REGION Network 55: STEP 1910~1940 : BDD CCV CHECK
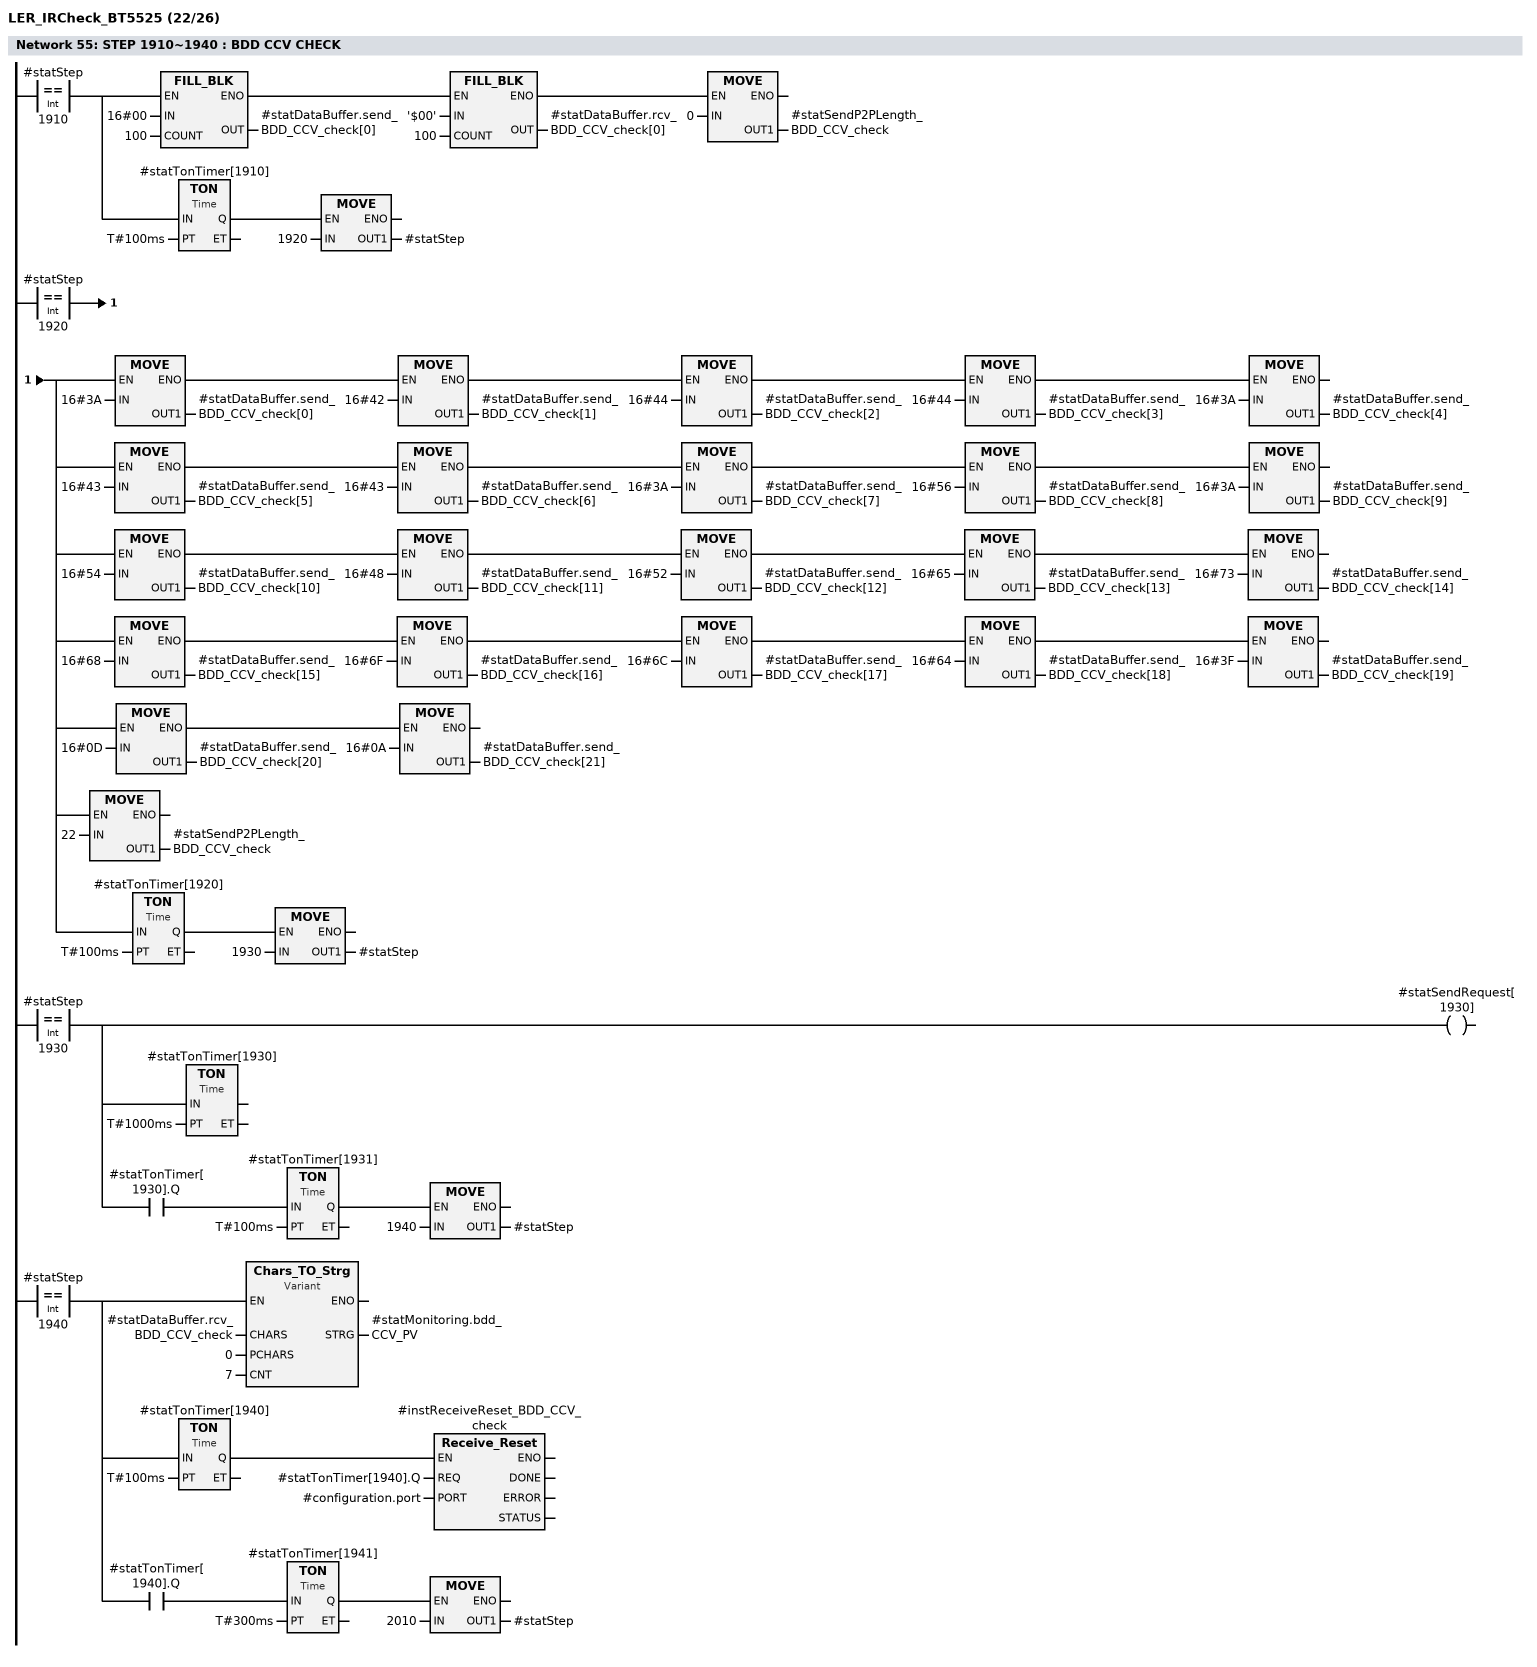
   RUNG wire#powerrail
      { S7_Templates := "SrcType := Int" } EQ_Contact(in1 := #statStep, in2 := 1910)
      wire#w1
      FillBlockI(in := 16#00, count := 100, out => #statDataBuffer.send_BDD_CCV_check[0])
      FillBlockI(in := '$00', count := 100, out => #statDataBuffer.rcv_BDD_CCV_check[0])
      Move(in := 0, out1 => #statSendP2PLength_BDD_CCV_check)
   END_RUNG
   RUNG wire#w1
      { S7_Templates := "time_type := Time" } #statTonTimer[1910].TON(pt := T#100ms, et =>)
      Move(in := 1920, out1 => #statStep)
   END_RUNG
   RUNG wire#powerrail
      { S7_Templates := "SrcType := Int" } EQ_Contact(in1 := #statStep, in2 := 1920)
      wire#w2
      Move(in := 16#3A, out1 => #statDataBuffer.send_BDD_CCV_check[0])
      Move(in := 16#42, out1 => #statDataBuffer.send_BDD_CCV_check[1])
      Move(in := 16#44, out1 => #statDataBuffer.send_BDD_CCV_check[2])
      Move(in := 16#44, out1 => #statDataBuffer.send_BDD_CCV_check[3])
      Move(in := 16#3A, out1 => #statDataBuffer.send_BDD_CCV_check[4])
   END_RUNG
   RUNG wire#w2
      Move(in := 16#43, out1 => #statDataBuffer.send_BDD_CCV_check[5])
      Move(in := 16#43, out1 => #statDataBuffer.send_BDD_CCV_check[6])
      Move(in := 16#3A, out1 => #statDataBuffer.send_BDD_CCV_check[7])
      Move(in := 16#56, out1 => #statDataBuffer.send_BDD_CCV_check[8])
      Move(in := 16#3A, out1 => #statDataBuffer.send_BDD_CCV_check[9])
   END_RUNG
   RUNG wire#w2
      Move(in := 16#54, out1 => #statDataBuffer.send_BDD_CCV_check[10])
      Move(in := 16#48, out1 => #statDataBuffer.send_BDD_CCV_check[11])
      Move(in := 16#52, out1 => #statDataBuffer.send_BDD_CCV_check[12])
      Move(in := 16#65, out1 => #statDataBuffer.send_BDD_CCV_check[13])
      Move(in := 16#73, out1 => #statDataBuffer.send_BDD_CCV_check[14])
   END_RUNG
   RUNG wire#w2
      Move(in := 16#68, out1 => #statDataBuffer.send_BDD_CCV_check[15])
      Move(in := 16#6F, out1 => #statDataBuffer.send_BDD_CCV_check[16])
      Move(in := 16#6C, out1 => #statDataBuffer.send_BDD_CCV_check[17])
      Move(in := 16#64, out1 => #statDataBuffer.send_BDD_CCV_check[18])
      Move(in := 16#3F, out1 => #statDataBuffer.send_BDD_CCV_check[19])
   END_RUNG
   RUNG wire#w2
      Move(in := 16#0D, out1 => #statDataBuffer.send_BDD_CCV_check[20])
      Move(in := 16#0A, out1 => #statDataBuffer.send_BDD_CCV_check[21])
   END_RUNG
   RUNG wire#w2
      Move(in := 22, out1 => #statSendP2PLength_BDD_CCV_check)
   END_RUNG
   RUNG wire#w2
      { S7_Templates := "time_type := Time" } #statTonTimer[1920].TON(pt := T#100ms, et =>)
      Move(in := 1930, out1 => #statStep)
   END_RUNG
   RUNG wire#powerrail
      { S7_Templates := "SrcType := Int" } EQ_Contact(in1 := #statStep, in2 := 1930)
      wire#w3
      Coil( #statSendRequest[1930] )
   END_RUNG
   RUNG wire#w3
      { S7_Templates := "time_type := Time" } #statTonTimer[1930].TON(pt := T#1000ms, et =>)
   END_RUNG
   RUNG wire#w3
      Contact( #statTonTimer[1930].Q )
      { S7_Templates := "time_type := Time" } #statTonTimer[1931].TON(pt := T#100ms, et =>)
      Move(in := 1940, out1 => #statStep)
   END_RUNG
   RUNG wire#powerrail
      { S7_Templates := "SrcType := Int" } EQ_Contact(in1 := #statStep, in2 := 1940)
      wire#w4
      { S7_Templates := "[ptr_type := Variant, str_type := String]" } Chars_TO_Strg(Chars := #statDataBuffer.rcv_BDD_CCV_check, pChars := 0, Cnt := 7, Strg => #statMonitoring.bdd_CCV_PV)
   END_RUNG
   RUNG wire#w4
      { S7_Templates := "time_type := Time" } #statTonTimer[1940].TON(pt := T#100ms, et =>)
      #instReceiveReset_BDD_CCV_check.Receive_Reset(REQ := #statTonTimer[1940].Q, PORT := #configuration.port, DONE =>, ERROR =>, STATUS =>)
   END_RUNG
   RUNG wire#w4
      Contact( #statTonTimer[1940].Q )
      { S7_Templates := "time_type := Time" } #statTonTimer[1941].TON(pt := T#300ms, et =>)
      Move(in := 2010, out1 => #statStep)
   END_RUNG
   // the same network as SCL:
   #_w1 := #statStep = 1910;
   IF #_w1 THEN
       FILL_BLK(IN := 16#00, COUNT := 100, OUT => #statDataBuffer.send_BDD_CCV_check[0]);
       FILL_BLK(IN := '$00', COUNT := 100, OUT => #statDataBuffer.rcv_BDD_CCV_check[0]);
       #statSendP2PLength_BDD_CCV_check := 0;
   END_IF;
   #statTonTimer[1910].TON(IN := #_w1, PT := T#100ms);
   IF #statTonTimer[1910].Q THEN #statStep := 1920; END_IF;
   #_w2 := #statStep = 1920;
   IF #_w2 THEN
       #statDataBuffer.send_BDD_CCV_check[0] := 16#3A;
       #statDataBuffer.send_BDD_CCV_check[1] := 16#42;
       #statDataBuffer.send_BDD_CCV_check[2] := 16#44;
       #statDataBuffer.send_BDD_CCV_check[3] := 16#44;
       #statDataBuffer.send_BDD_CCV_check[4] := 16#3A;
       #statDataBuffer.send_BDD_CCV_check[5] := 16#43;
       #statDataBuffer.send_BDD_CCV_check[6] := 16#43;
       #statDataBuffer.send_BDD_CCV_check[7] := 16#3A;
       #statDataBuffer.send_BDD_CCV_check[8] := 16#56;
       #statDataBuffer.send_BDD_CCV_check[9] := 16#3A;
       #statDataBuffer.send_BDD_CCV_check[10] := 16#54;
       #statDataBuffer.send_BDD_CCV_check[11] := 16#48;
       #statDataBuffer.send_BDD_CCV_check[12] := 16#52;
       #statDataBuffer.send_BDD_CCV_check[13] := 16#65;
       #statDataBuffer.send_BDD_CCV_check[14] := 16#73;
       #statDataBuffer.send_BDD_CCV_check[15] := 16#68;
       #statDataBuffer.send_BDD_CCV_check[16] := 16#6F;
       #statDataBuffer.send_BDD_CCV_check[17] := 16#6C;
       #statDataBuffer.send_BDD_CCV_check[18] := 16#64;
       #statDataBuffer.send_BDD_CCV_check[19] := 16#3F;
       #statDataBuffer.send_BDD_CCV_check[20] := 16#0D;
       #statDataBuffer.send_BDD_CCV_check[21] := 16#0A;
       #statSendP2PLength_BDD_CCV_check := 22;
   END_IF;
   #statTonTimer[1920].TON(IN := #_w2, PT := T#100ms);
   IF #statTonTimer[1920].Q THEN #statStep := 1930; END_IF;
   #statSendRequest[1930] := #statStep = 1930;
   #statTonTimer[1930].TON(IN := #statStep = 1930, PT := T#1000ms);
   #statTonTimer[1931].TON(IN := (#statStep = 1930) AND #statTonTimer[1930].Q, PT := T#100ms);
   IF #statTonTimer[1931].Q THEN #statStep := 1940; END_IF;
   #_w3 := #statStep = 1940;
   IF #_w3 THEN
       Chars_TO_Strg(Chars := #statDataBuffer.rcv_BDD_CCV_check,
                     pChars := 0,
                     Cnt := 7,
                     Strg => #statMonitoring.bdd_CCV_PV);
   END_IF;
   #statTonTimer[1940].TON(IN := #_w3, PT := T#100ms);
   IF #statTonTimer[1940].Q THEN
       #instReceiveReset_BDD_CCV_check(REQ := #statTonTimer[1940].Q, PORT := #configuration.port);   // Receive_Reset
   END_IF;
   #statTonTimer[1941].TON(IN := #_w3 AND #statTonTimer[1940].Q, PT := T#300ms);
   IF #statTonTimer[1941].Q THEN #statStep := 2010; END_IF;
END_REGION

REGION Network 56: STEP 2010~2030 : BDD CVV COMMAND
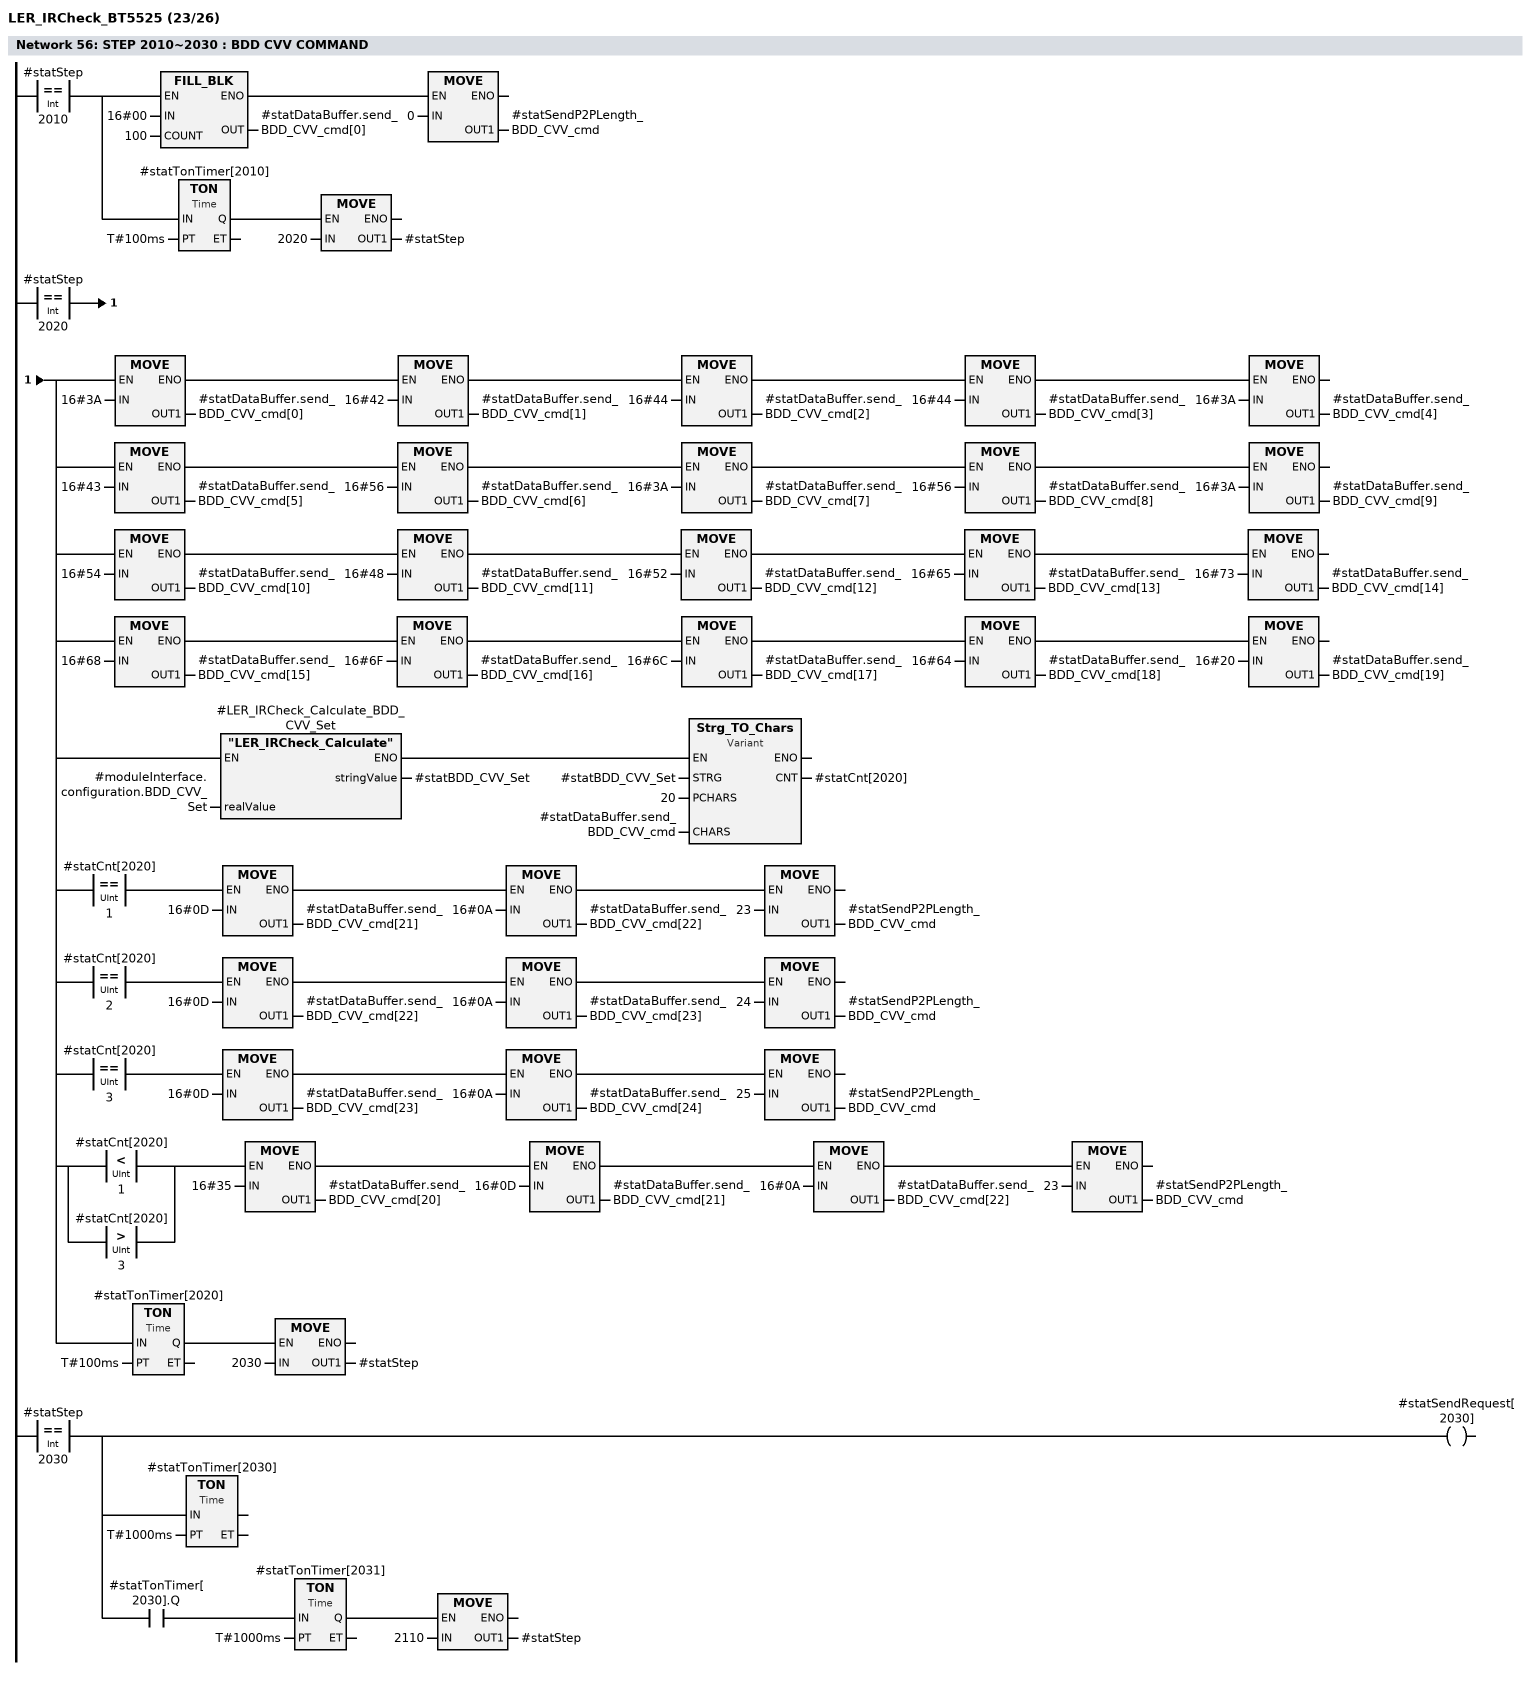
   RUNG wire#powerrail
      { S7_Templates := "SrcType := Int" } EQ_Contact(in1 := #statStep, in2 := 2010)
      wire#w1
      FillBlockI(in := 16#00, count := 100, out => #statDataBuffer.send_BDD_CVV_cmd[0])
      Move(in := 0, out1 => #statSendP2PLength_BDD_CVV_cmd)
   END_RUNG
   RUNG wire#w1
      { S7_Templates := "time_type := Time" } #statTonTimer[2010].TON(pt := T#100ms, et =>)
      Move(in := 2020, out1 => #statStep)
   END_RUNG
   RUNG wire#powerrail
      { S7_Templates := "SrcType := Int" } EQ_Contact(in1 := #statStep, in2 := 2020)
      wire#w2
      Move(in := 16#3A, out1 => #statDataBuffer.send_BDD_CVV_cmd[0])
      Move(in := 16#42, out1 => #statDataBuffer.send_BDD_CVV_cmd[1])
      Move(in := 16#44, out1 => #statDataBuffer.send_BDD_CVV_cmd[2])
      Move(in := 16#44, out1 => #statDataBuffer.send_BDD_CVV_cmd[3])
      Move(in := 16#3A, out1 => #statDataBuffer.send_BDD_CVV_cmd[4])
   END_RUNG
   RUNG wire#w2
      Move(in := 16#43, out1 => #statDataBuffer.send_BDD_CVV_cmd[5])
      Move(in := 16#56, out1 => #statDataBuffer.send_BDD_CVV_cmd[6])
      Move(in := 16#3A, out1 => #statDataBuffer.send_BDD_CVV_cmd[7])
      Move(in := 16#56, out1 => #statDataBuffer.send_BDD_CVV_cmd[8])
      Move(in := 16#3A, out1 => #statDataBuffer.send_BDD_CVV_cmd[9])
   END_RUNG
   RUNG wire#w2
      Move(in := 16#54, out1 => #statDataBuffer.send_BDD_CVV_cmd[10])
      Move(in := 16#48, out1 => #statDataBuffer.send_BDD_CVV_cmd[11])
      Move(in := 16#52, out1 => #statDataBuffer.send_BDD_CVV_cmd[12])
      Move(in := 16#65, out1 => #statDataBuffer.send_BDD_CVV_cmd[13])
      Move(in := 16#73, out1 => #statDataBuffer.send_BDD_CVV_cmd[14])
   END_RUNG
   RUNG wire#w2
      Move(in := 16#68, out1 => #statDataBuffer.send_BDD_CVV_cmd[15])
      Move(in := 16#6F, out1 => #statDataBuffer.send_BDD_CVV_cmd[16])
      Move(in := 16#6C, out1 => #statDataBuffer.send_BDD_CVV_cmd[17])
      Move(in := 16#64, out1 => #statDataBuffer.send_BDD_CVV_cmd[18])
      Move(in := 16#20, out1 => #statDataBuffer.send_BDD_CVV_cmd[19])
   END_RUNG
   RUNG wire#w2
      #LER_IRCheck_Calculate_BDD_CVV_Set(realValue := #moduleInterface.configuration.BDD_CVV_Set, stringValue => #statBDD_CVV_Set)
      { S7_Templates := "[ptr_type := Variant, strg_type := String]" } Strg_TO_Chars(Strg := #statBDD_CVV_Set, pChars := 20, Chars := #statDataBuffer.send_BDD_CVV_cmd, Cnt => #statCnt[2020])
   END_RUNG
   RUNG wire#w2
      { S7_Templates := "SrcType := UInt" } EQ_Contact(in1 := #statCnt[2020], in2 := 1)
      Move(in := 16#0D, out1 => #statDataBuffer.send_BDD_CVV_cmd[21])
      Move(in := 16#0A, out1 => #statDataBuffer.send_BDD_CVV_cmd[22])
      Move(in := 23, out1 => #statSendP2PLength_BDD_CVV_cmd)
   END_RUNG
   RUNG wire#w2
      { S7_Templates := "SrcType := UInt" } EQ_Contact(in1 := #statCnt[2020], in2 := 2)
      Move(in := 16#0D, out1 => #statDataBuffer.send_BDD_CVV_cmd[22])
      Move(in := 16#0A, out1 => #statDataBuffer.send_BDD_CVV_cmd[23])
      Move(in := 24, out1 => #statSendP2PLength_BDD_CVV_cmd)
   END_RUNG
   RUNG wire#w2
      { S7_Templates := "SrcType := UInt" } EQ_Contact(in1 := #statCnt[2020], in2 := 3)
      Move(in := 16#0D, out1 => #statDataBuffer.send_BDD_CVV_cmd[23])
      Move(in := 16#0A, out1 => #statDataBuffer.send_BDD_CVV_cmd[24])
      Move(in := 25, out1 => #statSendP2PLength_BDD_CVV_cmd)
   END_RUNG
   RUNG wire#w2
      { S7_Templates := "SrcType := UInt" } LT_Contact(in1 := #statCnt[2020], in2 := 1)
      wire#w3
      Move(in := 16#35, out1 => #statDataBuffer.send_BDD_CVV_cmd[20])
      Move(in := 16#0D, out1 => #statDataBuffer.send_BDD_CVV_cmd[21])
      Move(in := 16#0A, out1 => #statDataBuffer.send_BDD_CVV_cmd[22])
      Move(in := 23, out1 => #statSendP2PLength_BDD_CVV_cmd)
   END_RUNG
   RUNG wire#w2
      { S7_Templates := "SrcType := UInt" } GT_Contact(in1 := #statCnt[2020], in2 := 3)
   END_RUNG wire#w3
   RUNG wire#w2
      { S7_Templates := "time_type := Time" } #statTonTimer[2020].TON(pt := T#100ms, et =>)
      Move(in := 2030, out1 => #statStep)
   END_RUNG
   RUNG wire#powerrail
      { S7_Templates := "SrcType := Int" } EQ_Contact(in1 := #statStep, in2 := 2030)
      wire#w4
      Coil( #statSendRequest[2030] )
   END_RUNG
   RUNG wire#w4
      { S7_Templates := "time_type := Time" } #statTonTimer[2030].TON(pt := T#1000ms, et =>)
   END_RUNG
   RUNG wire#w4
      Contact( #statTonTimer[2030].Q )
      { S7_Templates := "time_type := Time" } #statTonTimer[2031].TON(pt := T#1000ms, et =>)
      Move(in := 2110, out1 => #statStep)
   END_RUNG
   // the same network as SCL:
   #_w1 := #statStep = 2010;
   IF #_w1 THEN
       FILL_BLK(IN := 16#00, COUNT := 100, OUT => #statDataBuffer.send_BDD_CVV_cmd[0]);
       #statSendP2PLength_BDD_CVV_cmd := 0;
   END_IF;
   #statTonTimer[2010].TON(IN := #_w1, PT := T#100ms);
   IF #statTonTimer[2010].Q THEN #statStep := 2020; END_IF;
   #_w2 := #statStep = 2020;
   IF #_w2 THEN
       #statDataBuffer.send_BDD_CVV_cmd[0] := 16#3A;
       #statDataBuffer.send_BDD_CVV_cmd[1] := 16#42;
       #statDataBuffer.send_BDD_CVV_cmd[2] := 16#44;
       #statDataBuffer.send_BDD_CVV_cmd[3] := 16#44;
       #statDataBuffer.send_BDD_CVV_cmd[4] := 16#3A;
       #statDataBuffer.send_BDD_CVV_cmd[5] := 16#43;
       #statDataBuffer.send_BDD_CVV_cmd[6] := 16#56;
       #statDataBuffer.send_BDD_CVV_cmd[7] := 16#3A;
       #statDataBuffer.send_BDD_CVV_cmd[8] := 16#56;
       #statDataBuffer.send_BDD_CVV_cmd[9] := 16#3A;
       #statDataBuffer.send_BDD_CVV_cmd[10] := 16#54;
       #statDataBuffer.send_BDD_CVV_cmd[11] := 16#48;
       #statDataBuffer.send_BDD_CVV_cmd[12] := 16#52;
       #statDataBuffer.send_BDD_CVV_cmd[13] := 16#65;
       #statDataBuffer.send_BDD_CVV_cmd[14] := 16#73;
       #statDataBuffer.send_BDD_CVV_cmd[15] := 16#68;
       #statDataBuffer.send_BDD_CVV_cmd[16] := 16#6F;
       #statDataBuffer.send_BDD_CVV_cmd[17] := 16#6C;
       #statDataBuffer.send_BDD_CVV_cmd[18] := 16#64;
       #statDataBuffer.send_BDD_CVV_cmd[19] := 16#20;
   END_IF;
   #LER_IRCheck_Calculate_BDD_CVV_Set(EN := #_w2,   // "LER_IRCheck_Calculate"
                           realValue := #moduleInterface.configuration.BDD_CVV_Set,
                           stringValue => #statBDD_CVV_Set,
                           ENO => #_w3);
   IF #_w3 THEN
       Strg_TO_Chars(Strg := #statBDD_CVV_Set,
                     pChars := 20,
                     Chars := #statDataBuffer.send_BDD_CVV_cmd,
                     Cnt => #statCnt[2020]);
   END_IF;
   IF #_w2 AND (#statCnt[2020] = 1) THEN
       #statDataBuffer.send_BDD_CVV_cmd[21] := 16#0D;
       #statDataBuffer.send_BDD_CVV_cmd[22] := 16#0A;
       #statSendP2PLength_BDD_CVV_cmd := 23;
   END_IF;
   IF #_w2 AND (#statCnt[2020] = 2) THEN
       #statDataBuffer.send_BDD_CVV_cmd[22] := 16#0D;
       #statDataBuffer.send_BDD_CVV_cmd[23] := 16#0A;
       #statSendP2PLength_BDD_CVV_cmd := 24;
   END_IF;
   IF #_w2 AND (#statCnt[2020] = 3) THEN
       #statDataBuffer.send_BDD_CVV_cmd[23] := 16#0D;
       #statDataBuffer.send_BDD_CVV_cmd[24] := 16#0A;
       #statSendP2PLength_BDD_CVV_cmd := 25;
   END_IF;
   IF #_w2 AND ((#statCnt[2020] < 1) OR (#statCnt[2020] > 3)) THEN
       #statDataBuffer.send_BDD_CVV_cmd[20] := 16#35;
       #statDataBuffer.send_BDD_CVV_cmd[21] := 16#0D;
       #statDataBuffer.send_BDD_CVV_cmd[22] := 16#0A;
       #statSendP2PLength_BDD_CVV_cmd := 23;
   END_IF;
   #statTonTimer[2020].TON(IN := #_w2, PT := T#100ms);
   IF #statTonTimer[2020].Q THEN #statStep := 2030; END_IF;
   #statSendRequest[2030] := #statStep = 2030;
   #statTonTimer[2030].TON(IN := #statStep = 2030, PT := T#1000ms);
   #statTonTimer[2031].TON(IN := (#statStep = 2030) AND #statTonTimer[2030].Q, PT := T#1000ms);
   IF #statTonTimer[2031].Q THEN #statStep := 2110; END_IF;
END_REGION

REGION Network 57: STEP 2110~2140 : BDD CVV CHECK
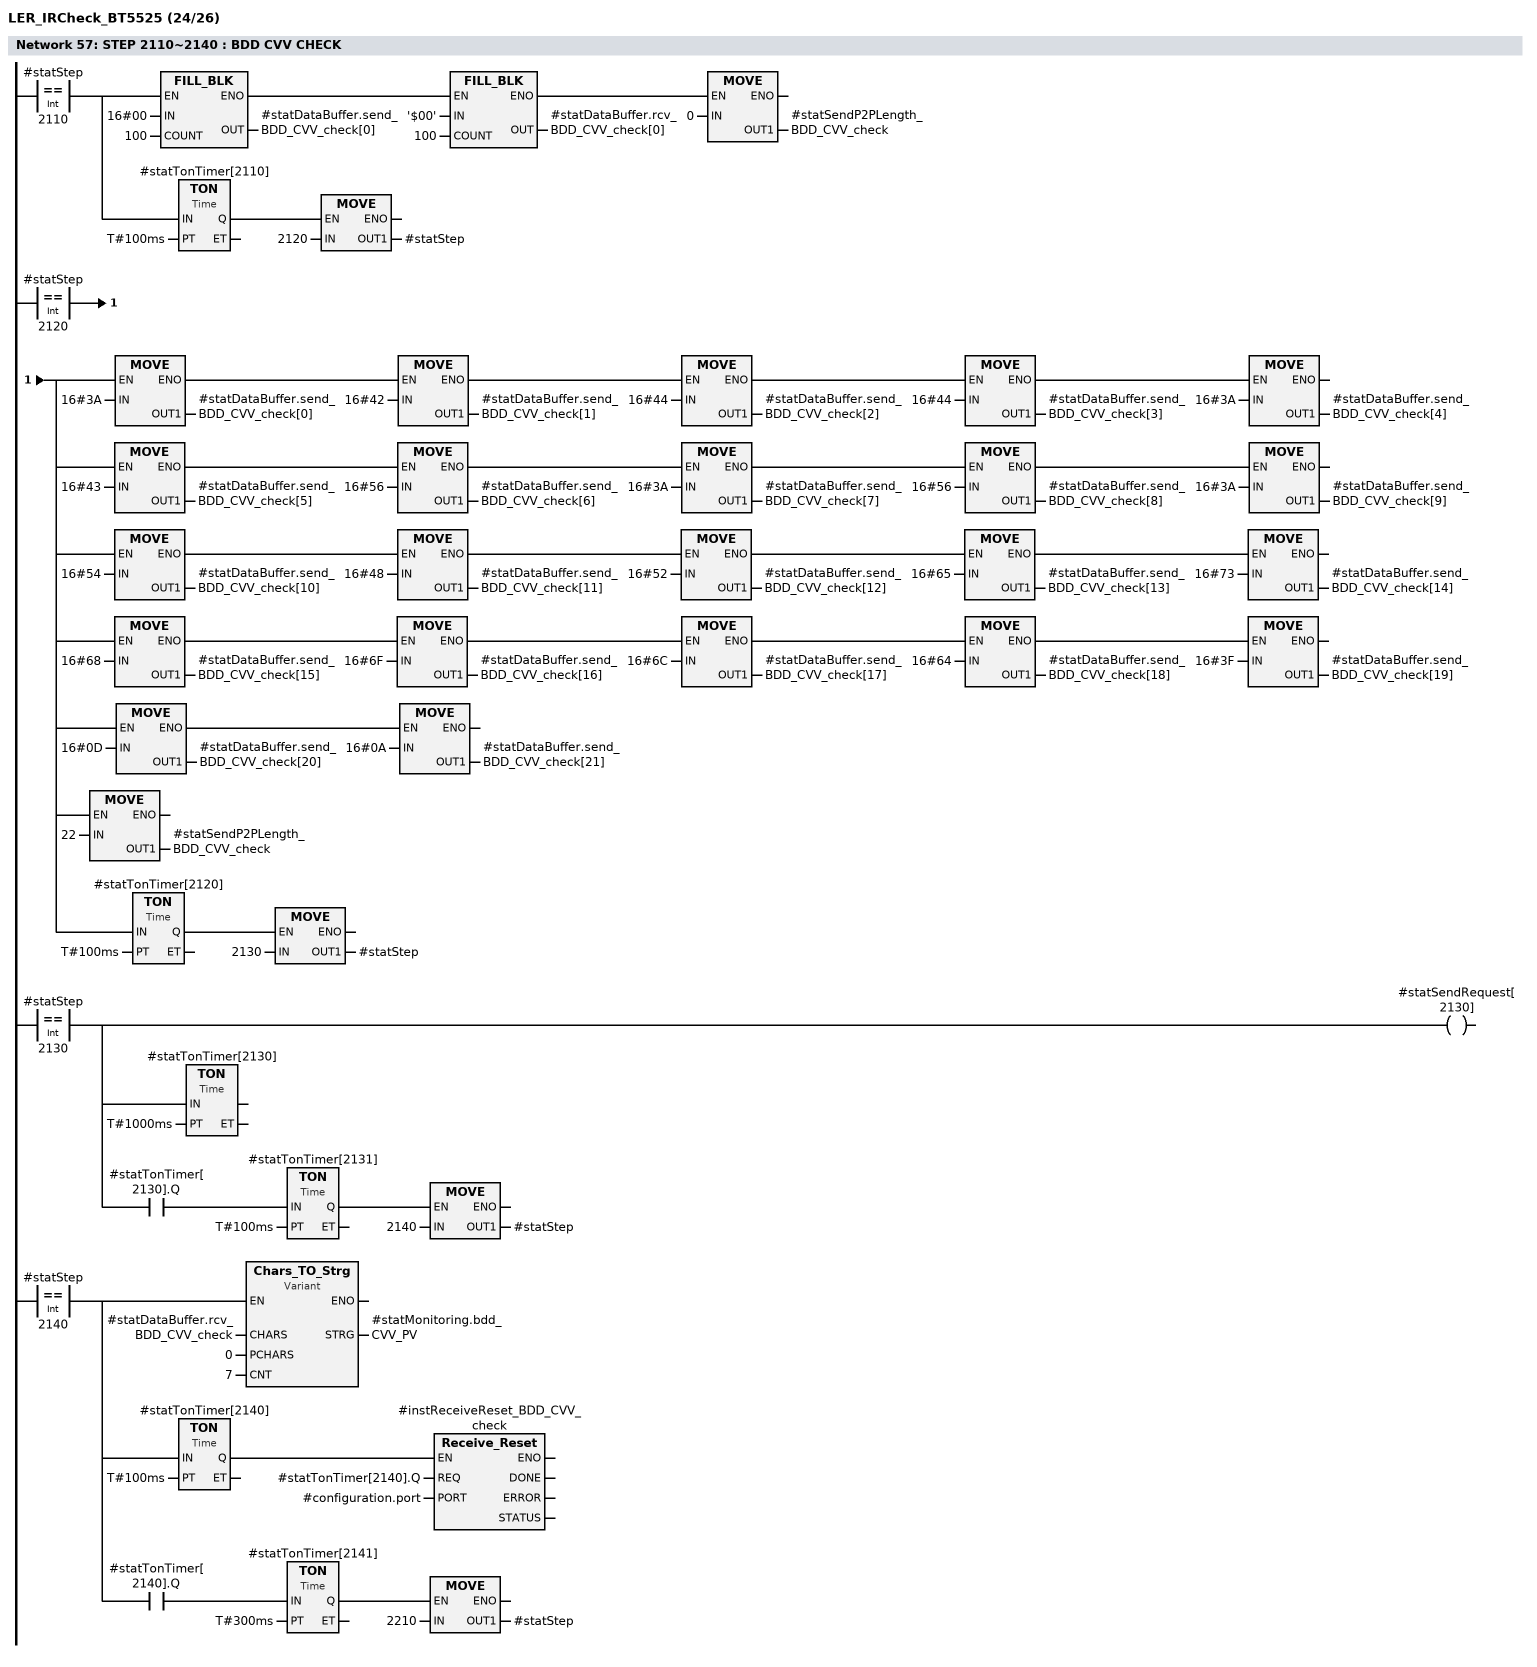
   RUNG wire#powerrail
      { S7_Templates := "SrcType := Int" } EQ_Contact(in1 := #statStep, in2 := 2110)
      wire#w1
      FillBlockI(in := 16#00, count := 100, out => #statDataBuffer.send_BDD_CVV_check[0])
      FillBlockI(in := '$00', count := 100, out => #statDataBuffer.rcv_BDD_CVV_check[0])
      Move(in := 0, out1 => #statSendP2PLength_BDD_CVV_check)
   END_RUNG
   RUNG wire#w1
      { S7_Templates := "time_type := Time" } #statTonTimer[2110].TON(pt := T#100ms, et =>)
      Move(in := 2120, out1 => #statStep)
   END_RUNG
   RUNG wire#powerrail
      { S7_Templates := "SrcType := Int" } EQ_Contact(in1 := #statStep, in2 := 2120)
      wire#w2
      Move(in := 16#3A, out1 => #statDataBuffer.send_BDD_CVV_check[0])
      Move(in := 16#42, out1 => #statDataBuffer.send_BDD_CVV_check[1])
      Move(in := 16#44, out1 => #statDataBuffer.send_BDD_CVV_check[2])
      Move(in := 16#44, out1 => #statDataBuffer.send_BDD_CVV_check[3])
      Move(in := 16#3A, out1 => #statDataBuffer.send_BDD_CVV_check[4])
   END_RUNG
   RUNG wire#w2
      Move(in := 16#43, out1 => #statDataBuffer.send_BDD_CVV_check[5])
      Move(in := 16#56, out1 => #statDataBuffer.send_BDD_CVV_check[6])
      Move(in := 16#3A, out1 => #statDataBuffer.send_BDD_CVV_check[7])
      Move(in := 16#56, out1 => #statDataBuffer.send_BDD_CVV_check[8])
      Move(in := 16#3A, out1 => #statDataBuffer.send_BDD_CVV_check[9])
   END_RUNG
   RUNG wire#w2
      Move(in := 16#54, out1 => #statDataBuffer.send_BDD_CVV_check[10])
      Move(in := 16#48, out1 => #statDataBuffer.send_BDD_CVV_check[11])
      Move(in := 16#52, out1 => #statDataBuffer.send_BDD_CVV_check[12])
      Move(in := 16#65, out1 => #statDataBuffer.send_BDD_CVV_check[13])
      Move(in := 16#73, out1 => #statDataBuffer.send_BDD_CVV_check[14])
   END_RUNG
   RUNG wire#w2
      Move(in := 16#68, out1 => #statDataBuffer.send_BDD_CVV_check[15])
      Move(in := 16#6F, out1 => #statDataBuffer.send_BDD_CVV_check[16])
      Move(in := 16#6C, out1 => #statDataBuffer.send_BDD_CVV_check[17])
      Move(in := 16#64, out1 => #statDataBuffer.send_BDD_CVV_check[18])
      Move(in := 16#3F, out1 => #statDataBuffer.send_BDD_CVV_check[19])
   END_RUNG
   RUNG wire#w2
      Move(in := 16#0D, out1 => #statDataBuffer.send_BDD_CVV_check[20])
      Move(in := 16#0A, out1 => #statDataBuffer.send_BDD_CVV_check[21])
   END_RUNG
   RUNG wire#w2
      Move(in := 22, out1 => #statSendP2PLength_BDD_CVV_check)
   END_RUNG
   RUNG wire#w2
      { S7_Templates := "time_type := Time" } #statTonTimer[2120].TON(pt := T#100ms, et =>)
      Move(in := 2130, out1 => #statStep)
   END_RUNG
   RUNG wire#powerrail
      { S7_Templates := "SrcType := Int" } EQ_Contact(in1 := #statStep, in2 := 2130)
      wire#w3
      Coil( #statSendRequest[2130] )
   END_RUNG
   RUNG wire#w3
      { S7_Templates := "time_type := Time" } #statTonTimer[2130].TON(pt := T#1000ms, et =>)
   END_RUNG
   RUNG wire#w3
      Contact( #statTonTimer[2130].Q )
      { S7_Templates := "time_type := Time" } #statTonTimer[2131].TON(pt := T#100ms, et =>)
      Move(in := 2140, out1 => #statStep)
   END_RUNG
   RUNG wire#powerrail
      { S7_Templates := "SrcType := Int" } EQ_Contact(in1 := #statStep, in2 := 2140)
      wire#w4
      { S7_Templates := "[ptr_type := Variant, str_type := String]" } Chars_TO_Strg(Chars := #statDataBuffer.rcv_BDD_CVV_check, pChars := 0, Cnt := 7, Strg => #statMonitoring.bdd_CVV_PV)
   END_RUNG
   RUNG wire#w4
      { S7_Templates := "time_type := Time" } #statTonTimer[2140].TON(pt := T#100ms, et =>)
      #instReceiveReset_BDD_CVV_check.Receive_Reset(REQ := #statTonTimer[2140].Q, PORT := #configuration.port, DONE =>, ERROR =>, STATUS =>)
   END_RUNG
   RUNG wire#w4
      Contact( #statTonTimer[2140].Q )
      { S7_Templates := "time_type := Time" } #statTonTimer[2141].TON(pt := T#300ms, et =>)
      Move(in := 2210, out1 => #statStep)
   END_RUNG
   // the same network as SCL:
   #_w1 := #statStep = 2110;
   IF #_w1 THEN
       FILL_BLK(IN := 16#00, COUNT := 100, OUT => #statDataBuffer.send_BDD_CVV_check[0]);
       FILL_BLK(IN := '$00', COUNT := 100, OUT => #statDataBuffer.rcv_BDD_CVV_check[0]);
       #statSendP2PLength_BDD_CVV_check := 0;
   END_IF;
   #statTonTimer[2110].TON(IN := #_w1, PT := T#100ms);
   IF #statTonTimer[2110].Q THEN #statStep := 2120; END_IF;
   #_w2 := #statStep = 2120;
   IF #_w2 THEN
       #statDataBuffer.send_BDD_CVV_check[0] := 16#3A;
       #statDataBuffer.send_BDD_CVV_check[1] := 16#42;
       #statDataBuffer.send_BDD_CVV_check[2] := 16#44;
       #statDataBuffer.send_BDD_CVV_check[3] := 16#44;
       #statDataBuffer.send_BDD_CVV_check[4] := 16#3A;
       #statDataBuffer.send_BDD_CVV_check[5] := 16#43;
       #statDataBuffer.send_BDD_CVV_check[6] := 16#56;
       #statDataBuffer.send_BDD_CVV_check[7] := 16#3A;
       #statDataBuffer.send_BDD_CVV_check[8] := 16#56;
       #statDataBuffer.send_BDD_CVV_check[9] := 16#3A;
       #statDataBuffer.send_BDD_CVV_check[10] := 16#54;
       #statDataBuffer.send_BDD_CVV_check[11] := 16#48;
       #statDataBuffer.send_BDD_CVV_check[12] := 16#52;
       #statDataBuffer.send_BDD_CVV_check[13] := 16#65;
       #statDataBuffer.send_BDD_CVV_check[14] := 16#73;
       #statDataBuffer.send_BDD_CVV_check[15] := 16#68;
       #statDataBuffer.send_BDD_CVV_check[16] := 16#6F;
       #statDataBuffer.send_BDD_CVV_check[17] := 16#6C;
       #statDataBuffer.send_BDD_CVV_check[18] := 16#64;
       #statDataBuffer.send_BDD_CVV_check[19] := 16#3F;
       #statDataBuffer.send_BDD_CVV_check[20] := 16#0D;
       #statDataBuffer.send_BDD_CVV_check[21] := 16#0A;
       #statSendP2PLength_BDD_CVV_check := 22;
   END_IF;
   #statTonTimer[2120].TON(IN := #_w2, PT := T#100ms);
   IF #statTonTimer[2120].Q THEN #statStep := 2130; END_IF;
   #statSendRequest[2130] := #statStep = 2130;
   #statTonTimer[2130].TON(IN := #statStep = 2130, PT := T#1000ms);
   #statTonTimer[2131].TON(IN := (#statStep = 2130) AND #statTonTimer[2130].Q, PT := T#100ms);
   IF #statTonTimer[2131].Q THEN #statStep := 2140; END_IF;
   #_w3 := #statStep = 2140;
   IF #_w3 THEN
       Chars_TO_Strg(Chars := #statDataBuffer.rcv_BDD_CVV_check,
                     pChars := 0,
                     Cnt := 7,
                     Strg => #statMonitoring.bdd_CVV_PV);
   END_IF;
   #statTonTimer[2140].TON(IN := #_w3, PT := T#100ms);
   IF #statTonTimer[2140].Q THEN
       #instReceiveReset_BDD_CVV_check(REQ := #statTonTimer[2140].Q, PORT := #configuration.port);   // Receive_Reset
   END_IF;
   #statTonTimer[2141].TON(IN := #_w3 AND #statTonTimer[2140].Q, PT := T#300ms);
   IF #statTonTimer[2141].Q THEN #statStep := 2210; END_IF;
END_REGION

REGION Network 58: STEP 2210~2230 : BDD CVI COMMAND
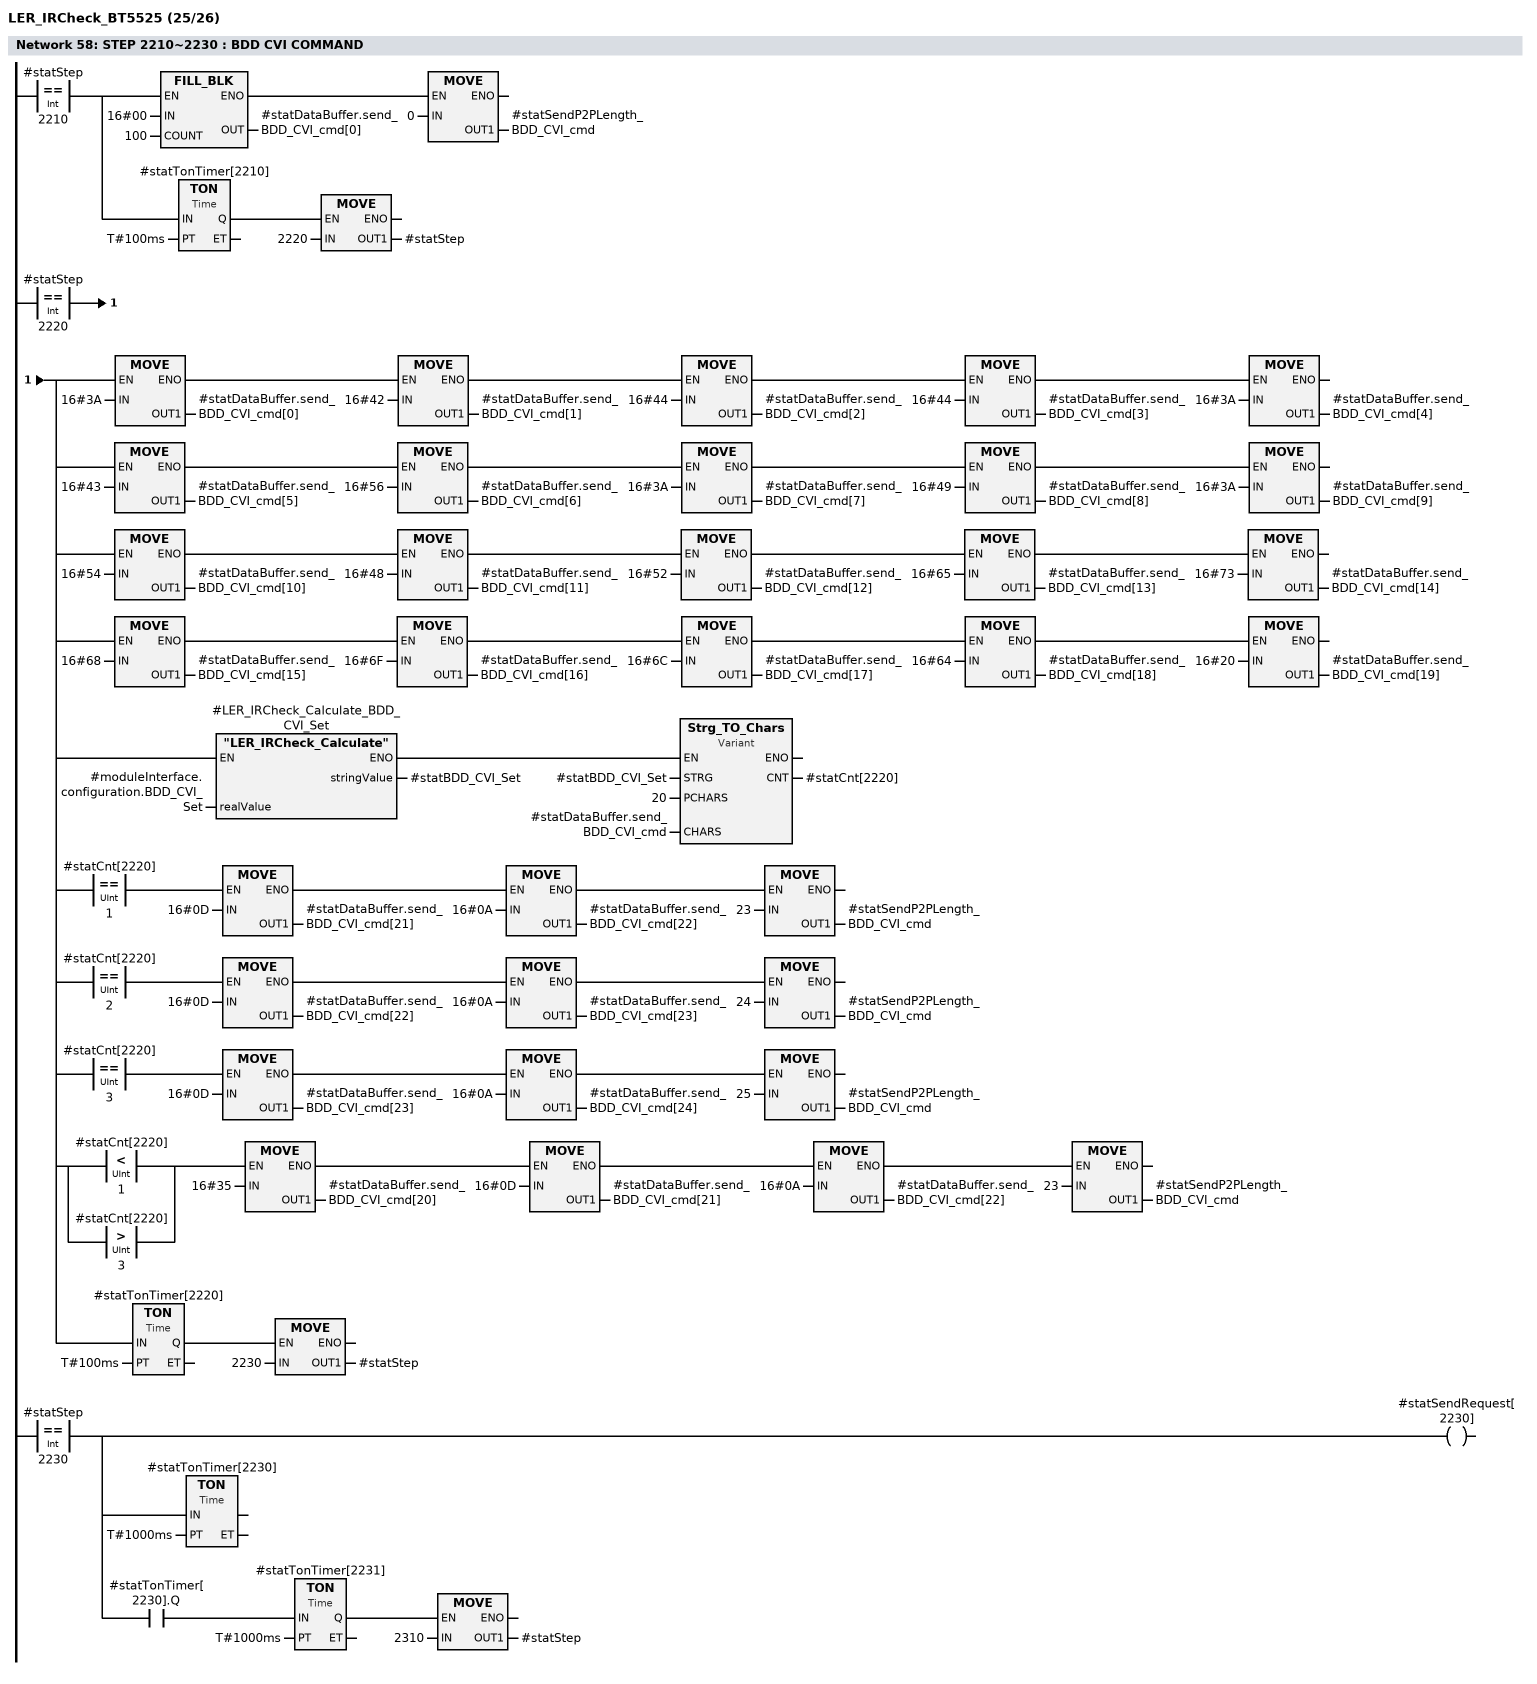
   RUNG wire#powerrail
      { S7_Templates := "SrcType := Int" } EQ_Contact(in1 := #statStep, in2 := 2210)
      wire#w1
      FillBlockI(in := 16#00, count := 100, out => #statDataBuffer.send_BDD_CVI_cmd[0])
      Move(in := 0, out1 => #statSendP2PLength_BDD_CVI_cmd)
   END_RUNG
   RUNG wire#w1
      { S7_Templates := "time_type := Time" } #statTonTimer[2210].TON(pt := T#100ms, et =>)
      Move(in := 2220, out1 => #statStep)
   END_RUNG
   RUNG wire#powerrail
      { S7_Templates := "SrcType := Int" } EQ_Contact(in1 := #statStep, in2 := 2220)
      wire#w2
      Move(in := 16#3A, out1 => #statDataBuffer.send_BDD_CVI_cmd[0])
      Move(in := 16#42, out1 => #statDataBuffer.send_BDD_CVI_cmd[1])
      Move(in := 16#44, out1 => #statDataBuffer.send_BDD_CVI_cmd[2])
      Move(in := 16#44, out1 => #statDataBuffer.send_BDD_CVI_cmd[3])
      Move(in := 16#3A, out1 => #statDataBuffer.send_BDD_CVI_cmd[4])
   END_RUNG
   RUNG wire#w2
      Move(in := 16#43, out1 => #statDataBuffer.send_BDD_CVI_cmd[5])
      Move(in := 16#56, out1 => #statDataBuffer.send_BDD_CVI_cmd[6])
      Move(in := 16#3A, out1 => #statDataBuffer.send_BDD_CVI_cmd[7])
      Move(in := 16#49, out1 => #statDataBuffer.send_BDD_CVI_cmd[8])
      Move(in := 16#3A, out1 => #statDataBuffer.send_BDD_CVI_cmd[9])
   END_RUNG
   RUNG wire#w2
      Move(in := 16#54, out1 => #statDataBuffer.send_BDD_CVI_cmd[10])
      Move(in := 16#48, out1 => #statDataBuffer.send_BDD_CVI_cmd[11])
      Move(in := 16#52, out1 => #statDataBuffer.send_BDD_CVI_cmd[12])
      Move(in := 16#65, out1 => #statDataBuffer.send_BDD_CVI_cmd[13])
      Move(in := 16#73, out1 => #statDataBuffer.send_BDD_CVI_cmd[14])
   END_RUNG
   RUNG wire#w2
      Move(in := 16#68, out1 => #statDataBuffer.send_BDD_CVI_cmd[15])
      Move(in := 16#6F, out1 => #statDataBuffer.send_BDD_CVI_cmd[16])
      Move(in := 16#6C, out1 => #statDataBuffer.send_BDD_CVI_cmd[17])
      Move(in := 16#64, out1 => #statDataBuffer.send_BDD_CVI_cmd[18])
      Move(in := 16#20, out1 => #statDataBuffer.send_BDD_CVI_cmd[19])
   END_RUNG
   RUNG wire#w2
      #LER_IRCheck_Calculate_BDD_CVI_Set(realValue := #moduleInterface.configuration.BDD_CVI_Set, stringValue => #statBDD_CVI_Set)
      { S7_Templates := "[ptr_type := Variant, strg_type := String]" } Strg_TO_Chars(Strg := #statBDD_CVI_Set, pChars := 20, Chars := #statDataBuffer.send_BDD_CVI_cmd, Cnt => #statCnt[2220])
   END_RUNG
   RUNG wire#w2
      { S7_Templates := "SrcType := UInt" } EQ_Contact(in1 := #statCnt[2220], in2 := 1)
      Move(in := 16#0D, out1 => #statDataBuffer.send_BDD_CVI_cmd[21])
      Move(in := 16#0A, out1 => #statDataBuffer.send_BDD_CVI_cmd[22])
      Move(in := 23, out1 => #statSendP2PLength_BDD_CVI_cmd)
   END_RUNG
   RUNG wire#w2
      { S7_Templates := "SrcType := UInt" } EQ_Contact(in1 := #statCnt[2220], in2 := 2)
      Move(in := 16#0D, out1 => #statDataBuffer.send_BDD_CVI_cmd[22])
      Move(in := 16#0A, out1 => #statDataBuffer.send_BDD_CVI_cmd[23])
      Move(in := 24, out1 => #statSendP2PLength_BDD_CVI_cmd)
   END_RUNG
   RUNG wire#w2
      { S7_Templates := "SrcType := UInt" } EQ_Contact(in1 := #statCnt[2220], in2 := 3)
      Move(in := 16#0D, out1 => #statDataBuffer.send_BDD_CVI_cmd[23])
      Move(in := 16#0A, out1 => #statDataBuffer.send_BDD_CVI_cmd[24])
      Move(in := 25, out1 => #statSendP2PLength_BDD_CVI_cmd)
   END_RUNG
   RUNG wire#w2
      { S7_Templates := "SrcType := UInt" } LT_Contact(in1 := #statCnt[2220], in2 := 1)
      wire#w3
      Move(in := 16#35, out1 => #statDataBuffer.send_BDD_CVI_cmd[20])
      Move(in := 16#0D, out1 => #statDataBuffer.send_BDD_CVI_cmd[21])
      Move(in := 16#0A, out1 => #statDataBuffer.send_BDD_CVI_cmd[22])
      Move(in := 23, out1 => #statSendP2PLength_BDD_CVI_cmd)
   END_RUNG
   RUNG wire#w2
      { S7_Templates := "SrcType := UInt" } GT_Contact(in1 := #statCnt[2220], in2 := 3)
   END_RUNG wire#w3
   RUNG wire#w2
      { S7_Templates := "time_type := Time" } #statTonTimer[2220].TON(pt := T#100ms, et =>)
      Move(in := 2230, out1 => #statStep)
   END_RUNG
   RUNG wire#powerrail
      { S7_Templates := "SrcType := Int" } EQ_Contact(in1 := #statStep, in2 := 2230)
      wire#w4
      Coil( #statSendRequest[2230] )
   END_RUNG
   RUNG wire#w4
      { S7_Templates := "time_type := Time" } #statTonTimer[2230].TON(pt := T#1000ms, et =>)
   END_RUNG
   RUNG wire#w4
      Contact( #statTonTimer[2230].Q )
      { S7_Templates := "time_type := Time" } #statTonTimer[2231].TON(pt := T#1000ms, et =>)
      Move(in := 2310, out1 => #statStep)
   END_RUNG
   // the same network as SCL:
   #_w1 := #statStep = 2210;
   IF #_w1 THEN
       FILL_BLK(IN := 16#00, COUNT := 100, OUT => #statDataBuffer.send_BDD_CVI_cmd[0]);
       #statSendP2PLength_BDD_CVI_cmd := 0;
   END_IF;
   #statTonTimer[2210].TON(IN := #_w1, PT := T#100ms);
   IF #statTonTimer[2210].Q THEN #statStep := 2220; END_IF;
   #_w2 := #statStep = 2220;
   IF #_w2 THEN
       #statDataBuffer.send_BDD_CVI_cmd[0] := 16#3A;
       #statDataBuffer.send_BDD_CVI_cmd[1] := 16#42;
       #statDataBuffer.send_BDD_CVI_cmd[2] := 16#44;
       #statDataBuffer.send_BDD_CVI_cmd[3] := 16#44;
       #statDataBuffer.send_BDD_CVI_cmd[4] := 16#3A;
       #statDataBuffer.send_BDD_CVI_cmd[5] := 16#43;
       #statDataBuffer.send_BDD_CVI_cmd[6] := 16#56;
       #statDataBuffer.send_BDD_CVI_cmd[7] := 16#3A;
       #statDataBuffer.send_BDD_CVI_cmd[8] := 16#49;
       #statDataBuffer.send_BDD_CVI_cmd[9] := 16#3A;
       #statDataBuffer.send_BDD_CVI_cmd[10] := 16#54;
       #statDataBuffer.send_BDD_CVI_cmd[11] := 16#48;
       #statDataBuffer.send_BDD_CVI_cmd[12] := 16#52;
       #statDataBuffer.send_BDD_CVI_cmd[13] := 16#65;
       #statDataBuffer.send_BDD_CVI_cmd[14] := 16#73;
       #statDataBuffer.send_BDD_CVI_cmd[15] := 16#68;
       #statDataBuffer.send_BDD_CVI_cmd[16] := 16#6F;
       #statDataBuffer.send_BDD_CVI_cmd[17] := 16#6C;
       #statDataBuffer.send_BDD_CVI_cmd[18] := 16#64;
       #statDataBuffer.send_BDD_CVI_cmd[19] := 16#20;
   END_IF;
   #LER_IRCheck_Calculate_BDD_CVI_Set(EN := #_w2,   // "LER_IRCheck_Calculate"
                           realValue := #moduleInterface.configuration.BDD_CVI_Set,
                           stringValue => #statBDD_CVI_Set,
                           ENO => #_w3);
   IF #_w3 THEN
       Strg_TO_Chars(Strg := #statBDD_CVI_Set,
                     pChars := 20,
                     Chars := #statDataBuffer.send_BDD_CVI_cmd,
                     Cnt => #statCnt[2220]);
   END_IF;
   IF #_w2 AND (#statCnt[2220] = 1) THEN
       #statDataBuffer.send_BDD_CVI_cmd[21] := 16#0D;
       #statDataBuffer.send_BDD_CVI_cmd[22] := 16#0A;
       #statSendP2PLength_BDD_CVI_cmd := 23;
   END_IF;
   IF #_w2 AND (#statCnt[2220] = 2) THEN
       #statDataBuffer.send_BDD_CVI_cmd[22] := 16#0D;
       #statDataBuffer.send_BDD_CVI_cmd[23] := 16#0A;
       #statSendP2PLength_BDD_CVI_cmd := 24;
   END_IF;
   IF #_w2 AND (#statCnt[2220] = 3) THEN
       #statDataBuffer.send_BDD_CVI_cmd[23] := 16#0D;
       #statDataBuffer.send_BDD_CVI_cmd[24] := 16#0A;
       #statSendP2PLength_BDD_CVI_cmd := 25;
   END_IF;
   IF #_w2 AND ((#statCnt[2220] < 1) OR (#statCnt[2220] > 3)) THEN
       #statDataBuffer.send_BDD_CVI_cmd[20] := 16#35;
       #statDataBuffer.send_BDD_CVI_cmd[21] := 16#0D;
       #statDataBuffer.send_BDD_CVI_cmd[22] := 16#0A;
       #statSendP2PLength_BDD_CVI_cmd := 23;
   END_IF;
   #statTonTimer[2220].TON(IN := #_w2, PT := T#100ms);
   IF #statTonTimer[2220].Q THEN #statStep := 2230; END_IF;
   #statSendRequest[2230] := #statStep = 2230;
   #statTonTimer[2230].TON(IN := #statStep = 2230, PT := T#1000ms);
   #statTonTimer[2231].TON(IN := (#statStep = 2230) AND #statTonTimer[2230].Q, PT := T#1000ms);
   IF #statTonTimer[2231].Q THEN #statStep := 2310; END_IF;
END_REGION

REGION Network 59: STEP 2310~2340 : BDD CVI CHECK
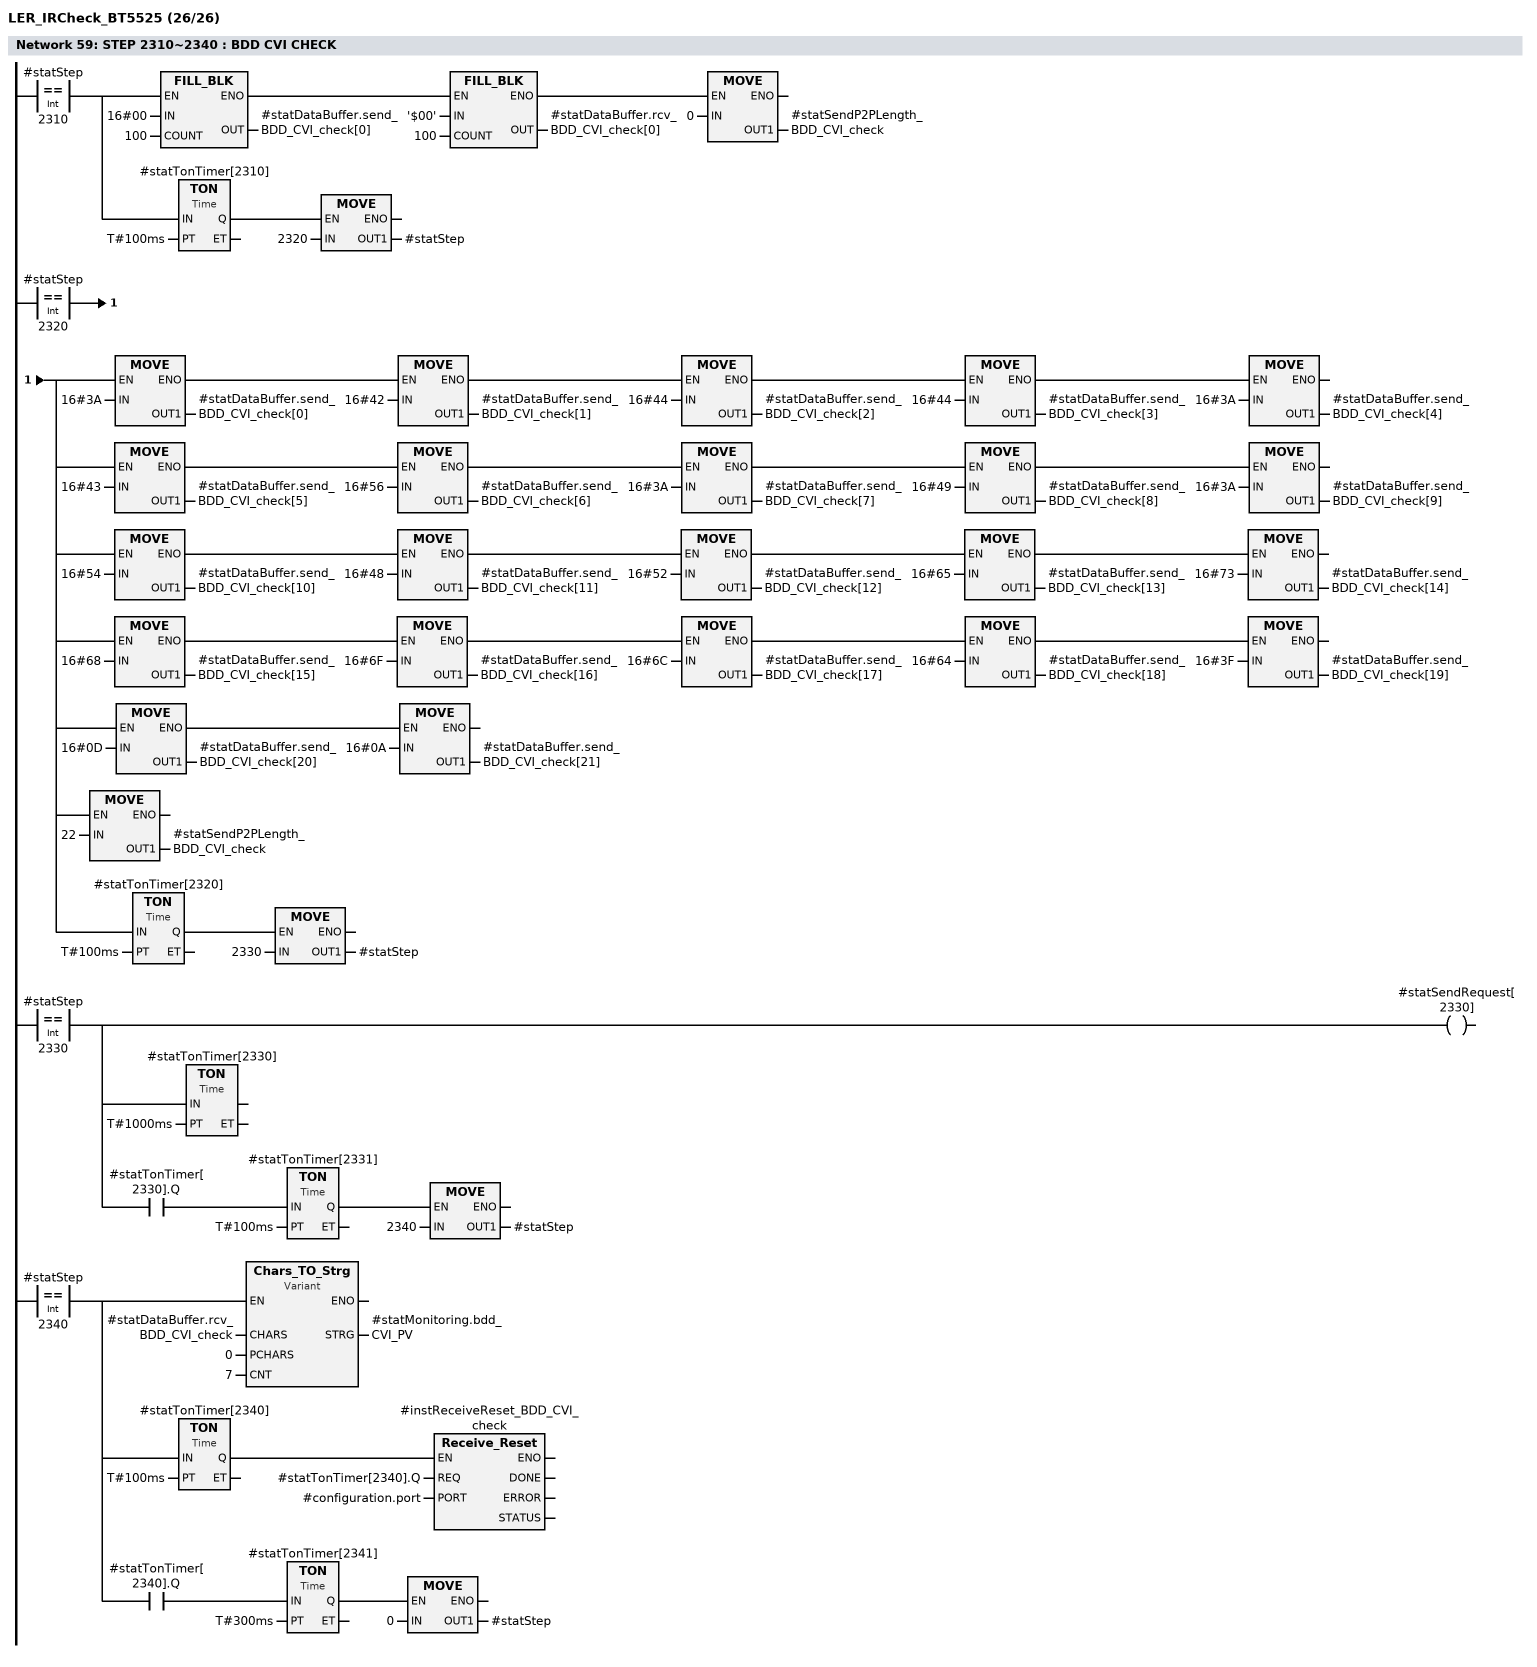
   RUNG wire#powerrail
      { S7_Templates := "SrcType := Int" } EQ_Contact(in1 := #statStep, in2 := 2310)
      wire#w1
      FillBlockI(in := 16#00, count := 100, out => #statDataBuffer.send_BDD_CVI_check[0])
      FillBlockI(in := '$00', count := 100, out => #statDataBuffer.rcv_BDD_CVI_check[0])
      Move(in := 0, out1 => #statSendP2PLength_BDD_CVI_check)
   END_RUNG
   RUNG wire#w1
      { S7_Templates := "time_type := Time" } #statTonTimer[2310].TON(pt := T#100ms, et =>)
      Move(in := 2320, out1 => #statStep)
   END_RUNG
   RUNG wire#powerrail
      { S7_Templates := "SrcType := Int" } EQ_Contact(in1 := #statStep, in2 := 2320)
      wire#w2
      Move(in := 16#3A, out1 => #statDataBuffer.send_BDD_CVI_check[0])
      Move(in := 16#42, out1 => #statDataBuffer.send_BDD_CVI_check[1])
      Move(in := 16#44, out1 => #statDataBuffer.send_BDD_CVI_check[2])
      Move(in := 16#44, out1 => #statDataBuffer.send_BDD_CVI_check[3])
      Move(in := 16#3A, out1 => #statDataBuffer.send_BDD_CVI_check[4])
   END_RUNG
   RUNG wire#w2
      Move(in := 16#43, out1 => #statDataBuffer.send_BDD_CVI_check[5])
      Move(in := 16#56, out1 => #statDataBuffer.send_BDD_CVI_check[6])
      Move(in := 16#3A, out1 => #statDataBuffer.send_BDD_CVI_check[7])
      Move(in := 16#49, out1 => #statDataBuffer.send_BDD_CVI_check[8])
      Move(in := 16#3A, out1 => #statDataBuffer.send_BDD_CVI_check[9])
   END_RUNG
   RUNG wire#w2
      Move(in := 16#54, out1 => #statDataBuffer.send_BDD_CVI_check[10])
      Move(in := 16#48, out1 => #statDataBuffer.send_BDD_CVI_check[11])
      Move(in := 16#52, out1 => #statDataBuffer.send_BDD_CVI_check[12])
      Move(in := 16#65, out1 => #statDataBuffer.send_BDD_CVI_check[13])
      Move(in := 16#73, out1 => #statDataBuffer.send_BDD_CVI_check[14])
   END_RUNG
   RUNG wire#w2
      Move(in := 16#68, out1 => #statDataBuffer.send_BDD_CVI_check[15])
      Move(in := 16#6F, out1 => #statDataBuffer.send_BDD_CVI_check[16])
      Move(in := 16#6C, out1 => #statDataBuffer.send_BDD_CVI_check[17])
      Move(in := 16#64, out1 => #statDataBuffer.send_BDD_CVI_check[18])
      Move(in := 16#3F, out1 => #statDataBuffer.send_BDD_CVI_check[19])
   END_RUNG
   RUNG wire#w2
      Move(in := 16#0D, out1 => #statDataBuffer.send_BDD_CVI_check[20])
      Move(in := 16#0A, out1 => #statDataBuffer.send_BDD_CVI_check[21])
   END_RUNG
   RUNG wire#w2
      Move(in := 22, out1 => #statSendP2PLength_BDD_CVI_check)
   END_RUNG
   RUNG wire#w2
      { S7_Templates := "time_type := Time" } #statTonTimer[2320].TON(pt := T#100ms, et =>)
      Move(in := 2330, out1 => #statStep)
   END_RUNG
   RUNG wire#powerrail
      { S7_Templates := "SrcType := Int" } EQ_Contact(in1 := #statStep, in2 := 2330)
      wire#w3
      Coil( #statSendRequest[2330] )
   END_RUNG
   RUNG wire#w3
      { S7_Templates := "time_type := Time" } #statTonTimer[2330].TON(pt := T#1000ms, et =>)
   END_RUNG
   RUNG wire#w3
      Contact( #statTonTimer[2330].Q )
      { S7_Templates := "time_type := Time" } #statTonTimer[2331].TON(pt := T#100ms, et =>)
      Move(in := 2340, out1 => #statStep)
   END_RUNG
   RUNG wire#powerrail
      { S7_Templates := "SrcType := Int" } EQ_Contact(in1 := #statStep, in2 := 2340)
      wire#w4
      { S7_Templates := "[ptr_type := Variant, str_type := String]" } Chars_TO_Strg(Chars := #statDataBuffer.rcv_BDD_CVI_check, pChars := 0, Cnt := 7, Strg => #statMonitoring.bdd_CVI_PV)
   END_RUNG
   RUNG wire#w4
      { S7_Templates := "time_type := Time" } #statTonTimer[2340].TON(pt := T#100ms, et =>)
      #instReceiveReset_BDD_CVI_check.Receive_Reset(REQ := #statTonTimer[2340].Q, PORT := #configuration.port, DONE =>, ERROR =>, STATUS =>)
   END_RUNG
   RUNG wire#w4
      Contact( #statTonTimer[2340].Q )
      { S7_Templates := "time_type := Time" } #statTonTimer[2341].TON(pt := T#300ms, et =>)
      Move(in := 0, out1 => #statStep)
   END_RUNG
   // the same network as SCL:
   #_w1 := #statStep = 2310;
   IF #_w1 THEN
       FILL_BLK(IN := 16#00, COUNT := 100, OUT => #statDataBuffer.send_BDD_CVI_check[0]);
       FILL_BLK(IN := '$00', COUNT := 100, OUT => #statDataBuffer.rcv_BDD_CVI_check[0]);
       #statSendP2PLength_BDD_CVI_check := 0;
   END_IF;
   #statTonTimer[2310].TON(IN := #_w1, PT := T#100ms);
   IF #statTonTimer[2310].Q THEN #statStep := 2320; END_IF;
   #_w2 := #statStep = 2320;
   IF #_w2 THEN
       #statDataBuffer.send_BDD_CVI_check[0] := 16#3A;
       #statDataBuffer.send_BDD_CVI_check[1] := 16#42;
       #statDataBuffer.send_BDD_CVI_check[2] := 16#44;
       #statDataBuffer.send_BDD_CVI_check[3] := 16#44;
       #statDataBuffer.send_BDD_CVI_check[4] := 16#3A;
       #statDataBuffer.send_BDD_CVI_check[5] := 16#43;
       #statDataBuffer.send_BDD_CVI_check[6] := 16#56;
       #statDataBuffer.send_BDD_CVI_check[7] := 16#3A;
       #statDataBuffer.send_BDD_CVI_check[8] := 16#49;
       #statDataBuffer.send_BDD_CVI_check[9] := 16#3A;
       #statDataBuffer.send_BDD_CVI_check[10] := 16#54;
       #statDataBuffer.send_BDD_CVI_check[11] := 16#48;
       #statDataBuffer.send_BDD_CVI_check[12] := 16#52;
       #statDataBuffer.send_BDD_CVI_check[13] := 16#65;
       #statDataBuffer.send_BDD_CVI_check[14] := 16#73;
       #statDataBuffer.send_BDD_CVI_check[15] := 16#68;
       #statDataBuffer.send_BDD_CVI_check[16] := 16#6F;
       #statDataBuffer.send_BDD_CVI_check[17] := 16#6C;
       #statDataBuffer.send_BDD_CVI_check[18] := 16#64;
       #statDataBuffer.send_BDD_CVI_check[19] := 16#3F;
       #statDataBuffer.send_BDD_CVI_check[20] := 16#0D;
       #statDataBuffer.send_BDD_CVI_check[21] := 16#0A;
       #statSendP2PLength_BDD_CVI_check := 22;
   END_IF;
   #statTonTimer[2320].TON(IN := #_w2, PT := T#100ms);
   IF #statTonTimer[2320].Q THEN #statStep := 2330; END_IF;
   #statSendRequest[2330] := #statStep = 2330;
   #statTonTimer[2330].TON(IN := #statStep = 2330, PT := T#1000ms);
   #statTonTimer[2331].TON(IN := (#statStep = 2330) AND #statTonTimer[2330].Q, PT := T#100ms);
   IF #statTonTimer[2331].Q THEN #statStep := 2340; END_IF;
   #_w3 := #statStep = 2340;
   IF #_w3 THEN
       Chars_TO_Strg(Chars := #statDataBuffer.rcv_BDD_CVI_check,
                     pChars := 0,
                     Cnt := 7,
                     Strg => #statMonitoring.bdd_CVI_PV);
   END_IF;
   #statTonTimer[2340].TON(IN := #_w3, PT := T#100ms);
   IF #statTonTimer[2340].Q THEN
       #instReceiveReset_BDD_CVI_check(REQ := #statTonTimer[2340].Q, PORT := #configuration.port);   // Receive_Reset
   END_IF;
   #statTonTimer[2341].TON(IN := #_w3 AND #statTonTimer[2340].Q, PT := T#300ms);
   IF #statTonTimer[2341].Q THEN #statStep := 0; END_IF;
END_REGION

REGION Network 60: ========================================== Mapping
END_REGION

REGION Network 61 (SCL): Output mapping
   REGION Output mapping

       #controlNode.monitoring := #moduleInterface.monitoring := #statMonitoring;

   END_REGION
END_REGION
END_FUNCTION_BLOCK
